// Mitsubishi GX Works2 project: 임시   PLC: Q02/Q02H

PROGRAM MAIN
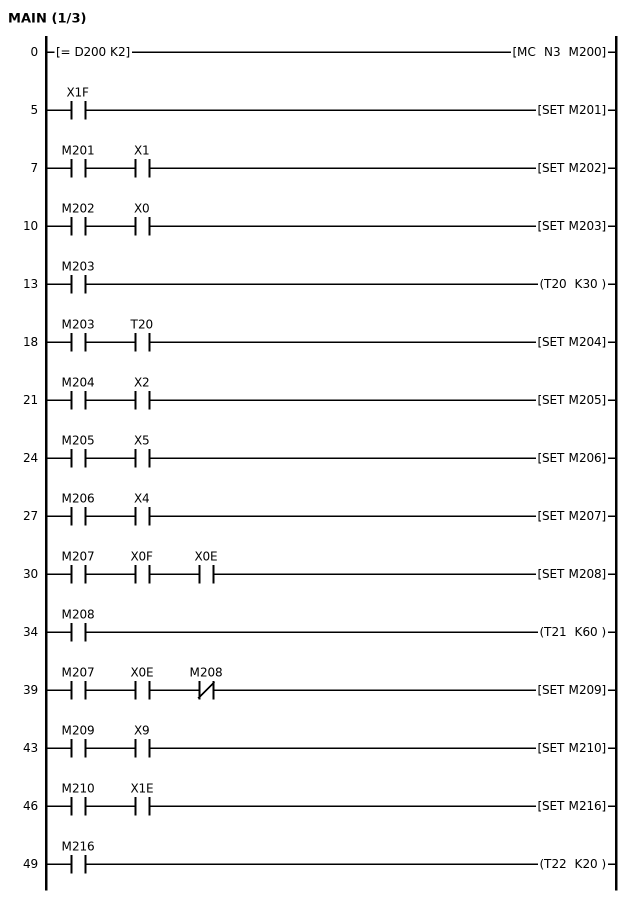
0     LD=     D200 K2
      MC      N3 M200
5     LD      X1F
      SET     M201
7     LD      M201
      AND     X1
      SET     M202
10    LD      M202
      AND     X0
      SET     M203
13    LD      M203
      OUT     T20 K30
18    LD      M203
      AND     T20
      SET     M204
21    LD      M204
      AND     X2
      SET     M205
24    LD      M205
      AND     X5
      SET     M206
27    LD      M206
      AND     X4
      SET     M207
30    LD      M207
      AND     X0F
      AND     X0E
      SET     M208
34    LD      M208
      OUT     T21 K60
39    LD      M207
      AND     X0E
      ANI     M208
      SET     M209
43    LD      M209
      AND     X9
      SET     M210
46    LD      M210
      AND     X1E
      SET     M216
49    LD      M216
      OUT     T22 K20
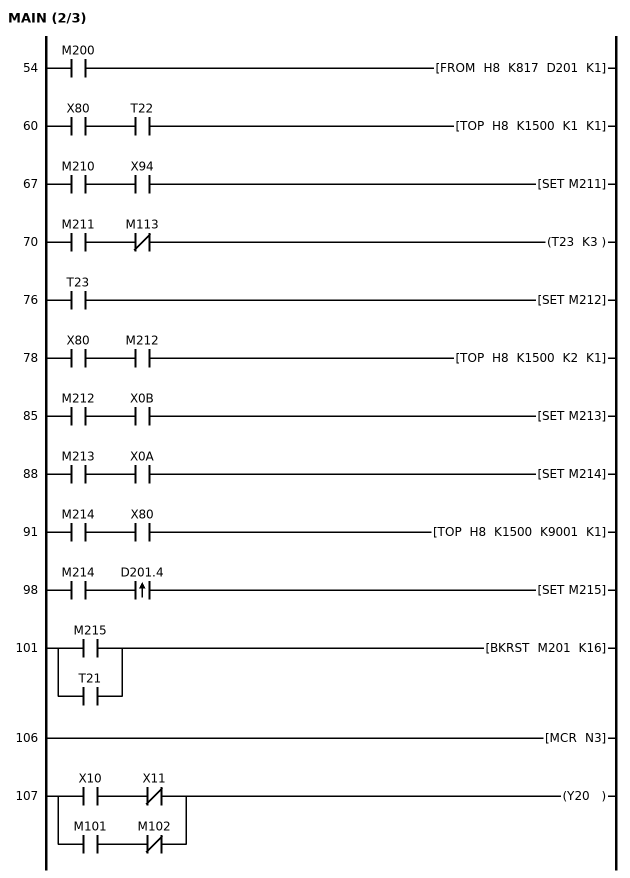
54    LD      M200
      FROM    H8 K817 D201 K1
60    LD      X80
      AND     T22
      TOP     H8 K1500 K1 K1
67    LD      M210
      AND     X94
      SET     M211
70    LD      M211
      ANI     M113
      OUT     T23 K3
76    LD      T23
      SET     M212
78    LD      X80
      AND     M212
      TOP     H8 K1500 K2 K1
85    LD      M212
      AND     X0B
      SET     M213
88    LD      M213
      AND     X0A
      SET     M214
91    LD      M214
      AND     X80
      TOP     H8 K1500 K9001 K1
98    LD      M214
      ANDP    D201.4
      SET     M215
101   LD      M215
      OR      T21
      BKRST   M201 K16
106   MCR     N3
107   LD      X10
      ANI     X11
      LD      M101
      ANI     M102
      ORB
      OUT     Y20
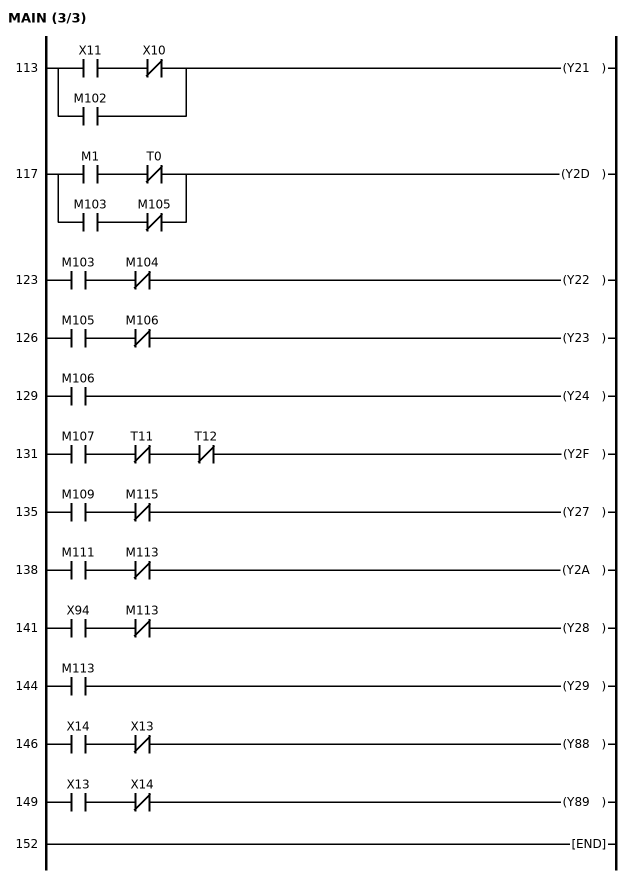
113   LD      X11
      ANI     X10
      OR      M102
      OUT     Y21
117   LD      M1
      ANI     T0
      LD      M103
      ANI     M105
      ORB
      OUT     Y2D
123   LD      M103
      ANI     M104
      OUT     Y22
126   LD      M105
      ANI     M106
      OUT     Y23
129   LD      M106
      OUT     Y24
131   LD      M107
      ANI     T11
      ANI     T12
      OUT     Y2F
135   LD      M109
      ANI     M115
      OUT     Y27
138   LD      M111
      ANI     M113
      OUT     Y2A
141   LD      X94
      ANI     M113
      OUT     Y28
144   LD      M113
      OUT     Y29
146   LD      X14
      ANI     X13
      OUT     Y88
149   LD      X13
      ANI     X14
      OUT     Y89
152   END
END_PROGRAM
